// TwinCAT 3 PLC project Prototype
// ProgramVersion: 3.1.4024.0
// libraries:
//   Tc2_Standard, * (Beckhoff Automation GmbH)
//   Tc2_System, * (Beckhoff Automation GmbH)
//   Tc3_Module, * (Beckhoff Automation GmbH)
// project tree:
//   / Class Diagram.TcCD (not stored), PlcTask.TcTTO (not stored)
//   Classes/ Circle.TcPOU, Disposable.TcPOU, I_Disposable.TcIO (not stored), Rectangle.TcPOU
//   Interfaces/ I_DrawableShape.TcIO (not stored)
//   POUs/ MAIN.TcPOU (not stored)
// real-time tasks:
//   TASK PlcTask: cycle T#10ms, priority 20, ADS port 350

// ---- Classes/Circle.TcPOU
{attribute 'enable_dynamic_creation'}
FUNCTION_BLOCK Circle EXTENDS Disposable IMPLEMENTS I_DrawableShape
VAR
	_radius: INT;
END_VAR

METHOD Clone : I_DrawableShape
VAR
	pCircle : POINTER TO Circle;	
END_VAR
pCircle := __NEW(Circle);
pCircle^.radius := radius;
Clone := pCircle^;
END_METHOD


METHOD Draw

VAR
	str : STRING;
END_VAR
str := TO_STRING(radius);
ADSLOGSTR(msgCtrlMask :=ADSLOG_MSGTYPE_HINT, msgFmtStr :='Draw circle with radius: %s', strArg := str);
END_METHOD

PROPERTY Radius : INT
GET
Radius := _radius;
END_GET
SET
_radius := Radius;
END_SET
END_PROPERTY

END_FUNCTION_BLOCK

// ---- Classes/Disposable.TcPOU
FUNCTION_BLOCK Disposable
VAR
END_VAR

METHOD PUBLIC Dispose
VAR_INPUT
END_VAR
__DELETE(THIS);
END_METHOD

END_FUNCTION_BLOCK

// ---- Classes/Rectangle.TcPOU
{attribute 'enable_dynamic_creation'}
FUNCTION_BLOCK Rectangle EXTENDS Disposable IMPLEMENTS I_DrawableShape
VAR
	_width: INT;
    _height: INT;
END_VAR

METHOD Clone : I_DrawableShape
VAR
	pRectangle : POINTER TO Rectangle;
END_VAR
pRectangle := __NEW(Rectangle);
pRectangle^.Width := Width;
pRectangle^.Height := Height;
Clone := pRectangle^;
END_METHOD

METHOD Draw
VAR
	str_width : STRING;
	str_height : STRING;
	str : STRING;
END_VAR
str_width := CONCAT(STR1 := 'width: ', STR2 := TO_STRING(Width));
str_height := CONCAT(STR1 := 'height: ', STR2 := TO_STRING(Height));
str := CONCAT(STR1 := str_width, STR2 := str_height);
ADSLOGSTR(msgCtrlMask := ADSLOG_MSGTYPE_HINT, msgFmtStr := 'Draw Rectangle with:  %s', strArg := str);
END_METHOD

PROPERTY PUBLIC Height : INT
GET
Height := _height;
END_GET
SET // PUBLIC
_height := Height;
END_SET
END_PROPERTY

PROPERTY PUBLIC Width : INT
GET
Width := _width;
END_GET
SET // PUBLIC
_width := Width;
END_SET
END_PROPERTY

END_FUNCTION_BLOCK
